TYPE ST_P_CHECK_TIMECONTROL :
STRUCT
	Barcode:			INT;
	ControlName:		STRING;
END_STRUCT
END_TYPE

(* stored: Version 1.1.0.1, ProductVersion 3.1.4024.10
   DUT ST_P_CHECK_TIMECONTROL: Id {af35da73-a09d-4c00-8ed6-657544ae6629} *)
